PROGRAM PRG_COM
VAR

END_VAR

(*Instanitate Serial port com function *)
fbSerialLineControl_SP1K2_PAX_PTM_01(
    Mode:= SERIALLINEMODE_EL6_22B,
    pComIn:= ADR(stComIn_SP1K2_PAX_PTM_01),
    pComOut:= ADR(stComOut_SP1K2_PAX_PTM_01),
    SizeComIn:= UINT_TO_INT(SIZEOF(stComIn_SP1K2_PAX_PTM_01)),
    TxBuffer:= SerialTXBuffer_SP1K2_PAX_PTM_01,
    RxBuffer:= SerialRXBuffer_SP1K2_PAX_PTM_01,
    Error=> ,
    ErrorID=> );

fbSerialLineControl_SP1K2_PAX_PTM_02(
    Mode:= SERIALLINEMODE_EL6_22B,
    pComIn:= ADR(stComIn_SP1K2_PAX_PTM_02),
    pComOut:= ADR(stComOut_SP1K2_PAX_PTM_02),
    SizeComIn:= UINT_TO_INT(SIZEOF(stComIn_SP1K2_PAX_PTM_02)),
    TxBuffer:= SerialTXBuffer_SP1K2_PAX_PTM_02,
    RxBuffer:= SerialRXBuffer_SP1K2_PAX_PTM_02,
    Error=> ,
    ErrorID=> );
	
fbSerialLineControl_LI3K2_K2B_OUT_PTM_01(
    Mode:= SERIALLINEMODE_EL6_22B,
    pComIn:= ADR(stComIn_LI3K2_K2B_OUT_PTM_01),
    pComOut:= ADR(stComOut_LI3K2_K2B_OUT_PTM_01),
    SizeComIn:= UINT_TO_INT(SIZEOF(stComIn_LI3K2_K2B_OUT_PTM_01)),
    TxBuffer:= SerialTXBuffer_LI3K2_K2B_OUT_PTM_01,
    RxBuffer:= SerialRXBuffer_LI3K2_K2B_OUT_PTM_01,
    Error=> ,
    ErrorID=> );
	
fbSerialLineControl_LI4K2_K2B_OUT_PTM_01(
    Mode:= SERIALLINEMODE_EL6_22B,
    pComIn:= ADR(stComIn_LI4K2_K2B_OUT_PTM_01),
    pComOut:= ADR(stComOut_LI4K2_K2B_OUT_PTM_01),
    SizeComIn:= UINT_TO_INT(SIZEOF(stComIn_LI4K2_K2B_OUT_PTM_01)),
    TxBuffer:= SerialTXBuffer_LI4K2_K2B_OUT_PTM_01,
    RxBuffer:= SerialRXBuffer_LI4K2_K2B_OUT_PTM_01,
    Error=> ,
    ErrorID=> );

END_PROGRAM

(* stored: Version 1.1.0.1, ProductVersion 3.1.4024.12
   POU PRG_COM: Id {b8dd9c68-f48c-4f7d-bf8f-7c6f0e748615}, SpecialFunc None *)
